{attribute 'qualified_only'}
{attribute 'strict'}
TYPE EExportState_t :
(
	eExportIdle := 0,
	eExportOpen,
	eExportGetLine,
	eExportWrite,
	eExportClose,
	eExportError
);
END_TYPE

(* stored: Version 1.1.0.1, ProductVersion 3.1.4024.12
   DUT EExportState_t: Id {e2b3d0d2-27df-4cd5-b2ce-fa95317235a2} *)
